// TIA Portal V18 program export: 1 tag tables, 0 data types, 2 data blocks, 2 code blocks (in call order from the OBs), 0 instance data blocks

VAR_GLOBAL   // PLC tag table "Tabella delle variabili standard"
END_VAR

DATA_BLOCK "Blocco_dati_1"
{ S7_Optimized_Access := 'TRUE' }
VERSION : 0.1
NON_RETAIN
   VAR 
      VARIABILE : Int;
      VARIABILE_1 : Int;
      VARIABILE_2 : Int;
      VARIABILE_3 : Int;
   END_VAR


BEGIN

END_DATA_BLOCK

DATA_BLOCK "Blocco_dati_2"
{ S7_Optimized_Access := 'TRUE' }
VERSION : 0.1
NON_RETAIN
   VAR 
      variabile : Bool;
      variabile_1 : Bool;
      variabile_2 : Bool;
      variabile_3 : Bool;
      variabile_4 : Bool;
      variabile_5 : Bool;
   END_VAR


BEGIN

END_DATA_BLOCK

ORGANIZATION_BLOCK "Main"   // OB1, LAD, ProgramCycle
TITLE = "Main Program Sweep (Cycle)"
{ S7_Optimized_Access := 'TRUE' }
VERSION : 0.1
// stored: AutoNumber true, IsIECCheckEnabled false, SetENOAutomatically false
   VAR_INPUT
      Initial_Call : Bool;   // Initial call of this OB
      Remanence : Bool;   // =True, if remanent data are available
   END_VAR
BEGIN
END_ORGANIZATION_BLOCK

FUNCTION_BLOCK "Blocco_1"   // FB1, LAD
{ S7_Optimized_Access := 'TRUE' }
VERSION : 0.1
// stored: AutoNumber true, IsIECCheckEnabled false, IsRetainMemResEnabled false, MemoryReserve 100, SetENOAutomatically false, UDAEnableTagReadback false
BEGIN
END_FUNCTION_BLOCK
